Fanuc KAREL source: ko00070.KL

-- PROVISIONAL review KL for V1013-1; original PC SHA256 cd6d03b619a752ee7a8747cf4c15414e2a40b33e4b3461e0053b7052919568cc
-- Incomplete behavior may be omitted. Consult companion uncertainty JSON. Do not deploy.
PROGRAM KO00070
%NOLOCKGROUP
BEGIN
  -- UNRESOLVED_PC offsets 5-12; opcodes 9D,23
  -- UNRESOLVED_PC offsets 17-66; opcodes 27,22,1C,27,49,7E,AD,22,31,7E,4A
  -- UNRESOLVED_PC offsets 71-75; opcodes 7F
END KO00070
